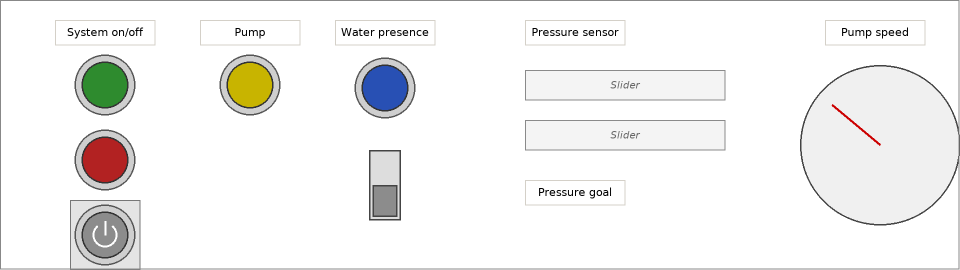
VISUALIZATION Visualization  // 960x270
    Lamp1 (70,50 70x70), variable: MAIN.System_on, style: Lamp-Lamp1-Green
    Slider (525,70 200x30), variable: MAIN.Pressure_sensor, scale 0..100
    PowerSwitch (70,200 70x70), variable: MAIN.System_switch, behaviour: TOGGLE, style: Switch-PowerSwitch-Gray
    Lamp1 (70,125 70x70), variable: MAIN.System_off, style: Lamp-Lamp1-Red
    Textfield (55,20 100x25), "System on/off"
    Textfield (200,20 100x25), "Pump"
    Lamp1 (215,50 70x70), variable: MAIN.Pump_on, style: Lamp-Lamp1-Yellow
    Lamp1 (350,53 70x70), variable: MAIN.Water_presence_light, style: Lamp-Lamp1-Blue
    Textfield (335,20 100x25), "Water presence"
    DipSwitch (350,150 70x70), variable: MAIN.Water_presence_sensor, behaviour: TOGGLE, style: Switch-DipSwitch-Gray
    Textfield (525,20 100x25), "Pressure sensor"
    Textfield (525,180 100x25), "Pressure goal"
    Slider (525,120 200x30), variable: MAIN.Pressure_Goal, scale 0..100
    Textfield (825,20 100x25), "Pump speed"
    Meter360 (800,65 160x160), value: MAIN.Pump_speed, style: Meter-Meter360-Gray, scale format: %.1f, scale 0..100
END_VISUALIZATION

(* stored: Version 1.1.0.1, ProductVersion 3.1.4024.12
   Visu Visualization: Id {effdf723-695d-42a4-8e58-f73c383b8695} *)
